INTERFACE I_AlarmTextList

METHOD GetAlarmText : STRING(ALARM_TEXT_SIZE)
VAR_INPUT
	nAlarmId : DINT;
END_VAR
END_METHOD

END_INTERFACE

(* stored: Version 1.1.0.1, ProductVersion 3.1.4024.15
   Itf I_AlarmTextList: Id {b866adc6-8f56-448e-b389-cdb43d8a333a}
   Method GetAlarmText: Id {9a0a98d0-7440-4c20-8b0f-4dff42afa739} *)
